FUNCTION_BLOCK ABSTRACT FB_Base IMPLEMENTS ITF_Base

VAR
	sName          										: STRING;
	uiId           										: UINT;
	
	              										
	bEnable        										: BOOL := TRUE;
	bInit          										: BOOL;
	bBusy          										: BOOL;
	bDone          										: BOOL;
	
	stError 													: ST_ErrorInfo;
	bError         										: BOOL;
	eErrorLevel												: E_ErrorLevel;
	uiErrorID													: UINT;
	sErrorOwner												: STRING;
	sErrorMessage  										: STRING;
END_VAR


IF NOT Init
  THEN Init := mInit();
END_IF

mVisu();

Enable := Enable;
IF NOT Enable 
	THEN 
		bBusy := FALSE;
		bDone := FALSE;
		RETURN; 
END_IF

mEnable();

PROPERTY Busy : bool
GET
Busy := bBusy;
END_GET
SET
bBusy := Busy;
END_SET
END_PROPERTY

PROPERTY Done : bool
GET
Done := bDone;
END_GET
SET
bDone := Done;
END_SET
END_PROPERTY

PROPERTY Enable : BOOL
GET
Enable := bEnable;
END_GET
SET
bEnable := Enable;
END_SET
END_PROPERTY

PROPERTY Error : bool
GET
Error := bError;
END_GET
SET
bError := Error;
END_SET
END_PROPERTY

PROPERTY ErrorID : UINT
GET
ErrorID := uiErrorID;
END_GET
SET
uiErrorID := ErrorID;
END_SET
END_PROPERTY

PROPERTY ErrorLevel : E_ErrorLevel
GET
ErrorLevel := eErrorLevel;
END_GET
SET
eErrorLevel := ErrorLevel;
END_SET
END_PROPERTY

PROPERTY ErrorMessage : STRING
GET
ErrorMessage := sErrorMessage;
END_GET
SET
sErrorMessage := ErrorMessage;
END_SET
END_PROPERTY

PROPERTY ErrorOwner : STRING
GET
ErrorOwner := sErrorOwner;
END_GET
SET
sErrorOwner := ErrorOwner;
END_SET
END_PROPERTY

//FB_Init ist immer implizit verfügbar und wird primär für die Initialisierung verwendet.
//Der Rückgabewert wird nicht ausgewertet. Für gezielte Einflussnahme können Sie
//die Methoden explizit deklarieren und darin mit dem Standard-Initialisierungscode 
//zusätzlichen Code bereitstellen. Sie können den Rückgabewert auswerten.
METHOD FB_Init: BOOL
VAR_INPUT    
	bInitRetains					: BOOL; 					// TRUE: Die Retain-Variablen werden initialisiert (Reset warm / Reset kalt)    
	bInCopyCode						: BOOL;  					// TRUE: Die Instanz wird danach in den Kopiercode kopiert (Online-Change)
	
	I_Name                : STRING;         //  Name
	I_ID                  : UINT;           // ID
//  I_itfOwner					  : ITF_Owner;      // owner 
END_VAR

Name          := I_Name;
ID            := I_ID;
END_METHOD

PROPERTY ID : UINT
GET
ID := uiID;
END_GET
SET
uiID := ID;
END_SET
END_PROPERTY

PROPERTY Init : BOOL
GET
Init := bInit;
END_GET
SET
bInit := Init;
END_SET
END_PROPERTY

METHOD mClearError : BOOL
VAR_INPUT
END_VAR

bError       		:= FALSE;
eErrorLevel  		:= E_ErrorLevel.NONE;
sErrorMessage   := '';
sErrorOwner  		:= '';

mClearError  		:= TRUE;
END_METHOD

METHOD mEnable : BOOL
VAR_INPUT
END_VAR

IF NOT bEnable THEN
    mEnable := FALSE;
    RETURN;
END_IF

IF bError THEN
    mEnable := FALSE;
    RETURN;
END_IF

mEnable := TRUE;
END_METHOD

METHOD mError : BOOL
VAR_INPUT
	I_sMessage   : STRING;
	I_eLevel		 : E_ErrorLevel;
	I_uiError		 : UINT;
END_VAR

stError.bActive				:= TRUE;
stError.eLevel				:= I_eLevel;
stError.uiErrorID			:= I_eLevel; 

stError.sOwner    		:= Name;
stError.sMessage			:= I_sMessage;

// Build full error message
stError.sFullMessage  := Concat(Name,':');
stError.sFullMessage  := Concat(stError.sFullMessage, I_sMessage);

// Error nur bei high oder critical Fehlern setzen
IF (I_eLevel = E_ErrorLevel.High)OR 
   (I_eLevel = E_ErrorLevel.Critical) 
	  	THEN
    		Error := TRUE;
END_IF

mError := TRUE;
END_METHOD

METHOD mInit : BOOL
VAR_INPUT

END_VAR

bBusy 					:= FALSE;
bDone 					:= FALSE;
bError 					:= FALSE;
sErrorMessage 	:= '';

mInit 					:= TRUE;
END_METHOD

METHOD mReset : BOOL
VAR_INPUT

END_VAR

bError 					:= FALSE;
bBusy 					:= FALSE;
bDone 					:= FALSE;
sErrorMessage 	:= '';

mReset 					:= TRUE;
END_METHOD

METHOD mVisu : BOOL
VAR_INPUT
END_VAR

mVisu:= TRUE;
END_METHOD

PROPERTY Name : string
GET
Name := sName;
END_GET
SET
sName := Name;
END_SET
END_PROPERTY

END_FUNCTION_BLOCK

(* stored: Version 1.1.0.1, ProductVersion 3.1.4026.18
   POU FB_Base: Id {b834a18a-92ee-42a2-95e8-764f580bbbef}, SpecialFunc None
   Folder 01 Properties: Id {5790059e-d17a-4094-b83c-c51da0ad590a}
   Folder 010 Error: Id {cc57b40f-bc69-496a-a242-392119a3fbc4}
   Folder 02 Methods: Id {1ddf855c-855f-4cab-bb1d-0e8290d5e41b}
   Property Busy: Id {4e93ede4-2583-440e-82cd-3ebd5d3c6673}
   Get Get: Id {74b8fd5a-a530-4365-a3d0-d5dfd4caa0ad}
   Set Set: Id {ad99bb6a-4889-4b2c-8d22-aae871c1edf0}
   Property Done: Id {c22f2f95-c83f-44ab-a967-0d2b231922e3}
   Get Get: Id {8ff8889d-7e46-4a97-a005-2964dcb813f0}
   Set Set: Id {4d09c58a-3a1e-4a6d-ad9e-9fb9f1c219db}
   Property Enable: Id {7593451e-2a4e-48d5-8158-cde01b66116d}
   Get Get: Id {ce3b6e85-e8f0-463a-a96b-c0fa51d59374}
   Set Set: Id {ed6a85ae-52ae-467d-a5da-492e73604bd4}
   Property Error: Id {4924a280-0be1-4edb-9696-4146f3ffac1c}
   Get Get: Id {6a5cde9d-1866-45f7-8066-0fb80f0c8369}
   Set Set: Id {23fa0463-603c-474d-bef4-9b3816af71aa}
   Property ErrorID: Id {5928cca3-c1f8-42ed-b513-0a877661f596}
   Get Get: Id {500dbc69-e34f-4975-8b6b-dc83623e8ef6}
   Set Set: Id {976fe0bd-91e9-442d-9f19-4d0f09047057}
   Property ErrorLevel: Id {f195f3e6-0351-4f68-86a3-e3dc5bd86f05}
   Get Get: Id {558024d4-a573-40c3-9376-34d41cbb8e1e}
   Set Set: Id {4a824867-8169-4e2d-9b58-fc82152c0962}
   Property ErrorMessage: Id {26b7aab4-54a0-4fbb-8ce3-4cb26fcfb03c}
   Get Get: Id {32609d22-1bfd-44b5-92ff-a201869fe3f3}
   Set Set: Id {f838be33-6957-42b7-a15f-8473a4b7b8f0}
   Property ErrorOwner: Id {2249a407-6057-4bd3-ad2b-8191f68d8bde}
   Get Get: Id {4e52ee2f-8b6a-49ee-b5ff-e0983ef4ebd9}
   Set Set: Id {feb04ec4-85da-4029-86f9-32c819f20771}
   Method FB_Init: Id {149da957-1655-4e71-bdf4-dda83c59d4da}
   Property ID: Id {e5dc53a9-c3da-4ce2-85f4-2d2964df44e1}
   Get Get: Id {ae6a7782-c6a2-40a9-a812-57110336a9a9}
   Set Set: Id {cba7ebe4-90d6-494b-acfb-2deb84bb1d02}
   Property Init: Id {1fe9019d-f4c9-4a94-a3f1-811245f6dd83}
   Get Get: Id {0a4395c4-7ded-4389-83b0-9e8401455921}
   Set Set: Id {e39de7f1-5a87-46b8-8af6-28dc0f0740f0}
   Method mClearError: Id {c87b6c47-8da3-4b17-8289-16b94d7267e4}
   Method mEnable: Id {5ac26998-73d7-403c-92b8-3bfaf4bc5e70}
   Method mError: Id {ee1ebbbd-87be-4bbf-887f-72641b7ae4ae}
   Method mInit: Id {85ac23e9-5592-4108-b8d8-74958e7f3617}
   Method mReset: Id {aeb080ea-8eb0-4963-90f8-ddb74f05dd39}
   Method mVisu: Id {1111107a-3623-4d0d-a6e5-8e620036109e}
   Property Name: Id {f9504863-6599-48cb-8f38-c5a44834f50f}
   Get Get: Id {af3df418-e680-40d5-8e46-9655428744e8}
   Set Set: Id {782ec1bd-9532-4aec-a974-ccfca001f4fa} *)
